(* Schneider Machine Expert - Basic project VirtualPLC_Dynamic, file version 2.6.0.0 *)
(* ProjectInformations: Name=Capstone D-03 *)
(* UserInformations: LastName=D-03, FirstName=Capstone Project *)

HARDWARE
  Cpu 0: TM221ME16R/G
  ModuleExtensionObject 0: TM3DQ8R/G
  ModuleExtensionObject 1: TM3AI8/G
  ModuleExtensionObject 2: TM3AI8/G
  EthernetConfiguration: NetworkName=M221, IpAllocationMode=FixedAddress, IpAddress=192.168.100.195, SubnetMask=255.255.255.0
  SerialLineConfiguration: Baud=Baud19200, Parity=ParityEven, DataBits=DataBits8, StopBits=StopBits1, PhysicalMedium=PhysicalMediumRs485, SlaveId=1, Addressing=SlaveAddressing
  MastTask: UsePeriodScanMode=false, PeriodScan=100
  FastTask: Period=255
  CpuBehavior: StartingMode=StartAsPreviousState, AutoSaveRamOnEeprom=true, WatchdogPeriod=250

SYMBOLS  (address, symbol, comment, settings)
  %M0       READ_GEN1
  %M1       READ_GEN2
  %M2       READ_GEN3
  %M3       READ_GEN4
  %M10      STATUS_GEN_1A_75MW
  %M11      STATUS_GEN_1B_25_MW
  %M12      STATUS_GEN_1B_75MW
  %M13      STATUS_GEN_2B_25_MW
  %M21      L101
  %M22      L201
  %M23      L303
  %M24      L304
  %M25      L305
  %M26      L401
  %M31      L301
  %M32      L302
  %M33      L402
  %M41      L403
  %M42      L404
  %M43      L405
  %M50      CONTROL_GEN1
  %M51      CONTROL_GEN2
  %M52      CONTROL_GEN3
  %M53      CONTROL_GEN4
  %M60      READ_LOAD1
  %M61      READ_LOAD2
  %M62      READ_LOAD3
  %M63      READ_LOAD4
  %M64      READ_LOAD5
  %M65      READ_LOAD6
  %M66      READ_LOAD7
  %M67      READ_LOAD8
  %M68      READ_LOAD9
  %M69      READ_LOAD10
  %M70      READ_LOAD11
  %M71      READ_LOAD12
  %MW0      SENSOR_LOAD1
  %MW1      SENSOR_LOAD2
  %MW2      SENSOR_LOAD3
  %MW3      SENSOR_LOAD4
  %MW4      SENSOR_LOAD5
  %MW5      SENSOR_LOAD6
  %MW6      SENSOR_LOAD7
  %MW7      SENSOR_LOAD8
  %MW8      SENSOR_LOAD9
  %MW9      SENSOR_LOAD10
  %MW10     SENSOR_LOAD11
  %MW11     SENSOR_LOAD12
  %MW20     JAM
  %MW21     MENIT
  %MW30     SENSOR_GEN1  "PLTA"
  %MW31     SENSOR_GEN2  "PLTS"
  %MW32     SENSOR_GEN3  "PLTGU"
  %MW33     SENSOR_GEN4  "PLTB"
  %MW54     FREQ
  %Q0.0     COIL_GEN1
  %Q0.1     COIL_GEN2
  %Q0.2     COIL_GEN3
  %Q0.3     COIL_GEN4
  %Q0.4     COIL_LOAD1
  %Q0.5     COIL_LOAD2
  %Q0.6     COIL_LOAD3
  %Q0.7     COIL_LOAD4
  %IW0.0    GEN_1_SIM  [Type=Type_0_10V, Scope=Scope_Normal, Minimum=0, Maximum=1000]
  %Q1.0     COIL_LOAD5
  %Q1.1     COIL_LOAD6
  %Q1.2     COIL_LOAD7
  %Q1.3     COIL_LOAD8
  %Q1.4     COIL_LOAD9
  %Q1.5     COIL_LOAD10
  %Q1.6     COIL_LOAD11
  %Q1.7     COIL_LOAD12

POU New POU
  (* SectionNumber=1 *)

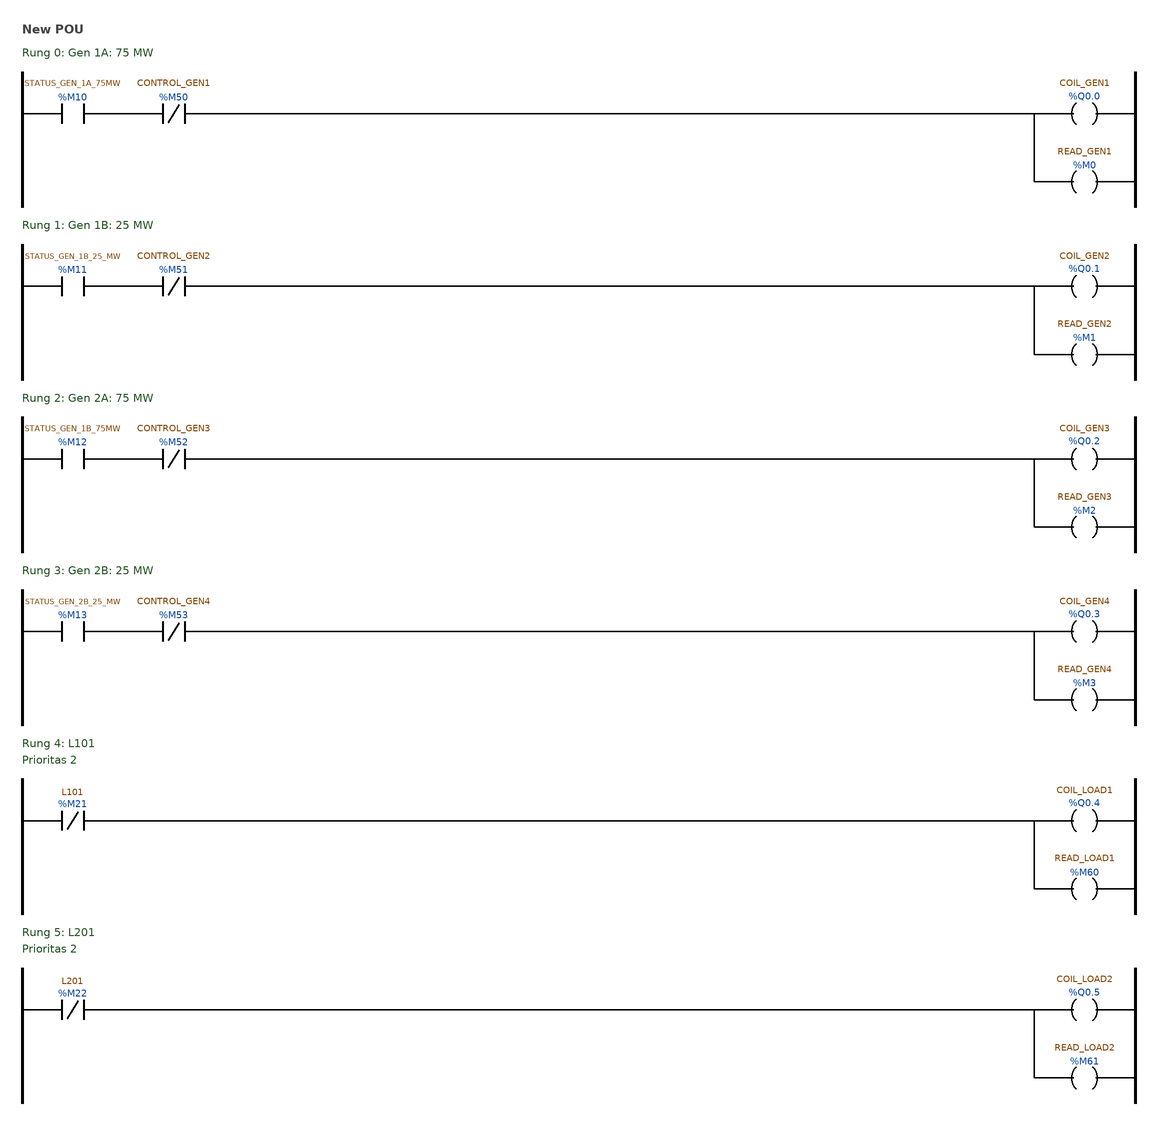

// Rung 0: Gen 1A: 75 MW
  LD %M10                 (* STATUS_GEN_1A_75MW *)
  ANDN %M50               (* CONTROL_GEN1 *)
  ST %Q0.0                (* COIL_GEN1 *)
  ST %M0                  (* READ_GEN1 *)
  // as ST:
  //   COIL_GEN1 := STATUS_GEN_1A_75MW AND NOT CONTROL_GEN1;
  //   READ_GEN1 := STATUS_GEN_1A_75MW AND NOT CONTROL_GEN1;

// Rung 1: Gen 1B: 25 MW
  LD %M11                 (* STATUS_GEN_1B_25_MW *)
  ANDN %M51               (* CONTROL_GEN2 *)
  ST %Q0.1                (* COIL_GEN2 *)
  ST %M1                  (* READ_GEN2 *)
  // as ST:
  //   COIL_GEN2 := STATUS_GEN_1B_25_MW AND NOT CONTROL_GEN2;
  //   READ_GEN2 := STATUS_GEN_1B_25_MW AND NOT CONTROL_GEN2;

// Rung 2: Gen 2A: 75 MW
  LD %M12                 (* STATUS_GEN_1B_75MW *)
  ANDN %M52               (* CONTROL_GEN3 *)
  ST %Q0.2                (* COIL_GEN3 *)
  ST %M2                  (* READ_GEN3 *)
  // as ST:
  //   COIL_GEN3 := STATUS_GEN_1B_75MW AND NOT CONTROL_GEN3;
  //   READ_GEN3 := STATUS_GEN_1B_75MW AND NOT CONTROL_GEN3;

// Rung 3: Gen 2B: 25 MW
  LD %M13                 (* STATUS_GEN_2B_25_MW *)
  ANDN %M53               (* CONTROL_GEN4 *)
  ST %Q0.3                (* COIL_GEN4 *)
  ST %M3                  (* READ_GEN4 *)
  // as ST:
  //   COIL_GEN4 := STATUS_GEN_2B_25_MW AND NOT CONTROL_GEN4;
  //   READ_GEN4 := STATUS_GEN_2B_25_MW AND NOT CONTROL_GEN4;

// Rung 4: L101
// Prioritas 2
  LDN %M21                (* L101 *)
  ST %Q0.4                (* COIL_LOAD1 *)
  ST %M60                 (* READ_LOAD1 *)
  // as ST:
  //   COIL_LOAD1 := NOT L101;
  //   READ_LOAD1 := NOT L101;

// Rung 5: L201
// Prioritas 2
  LDN %M22                (* L201 *)
  ST %Q0.5                (* COIL_LOAD2 *)
  ST %M61                 (* READ_LOAD2 *)
  // as ST:
  //   COIL_LOAD2 := NOT L201;
  //   READ_LOAD2 := NOT L201;

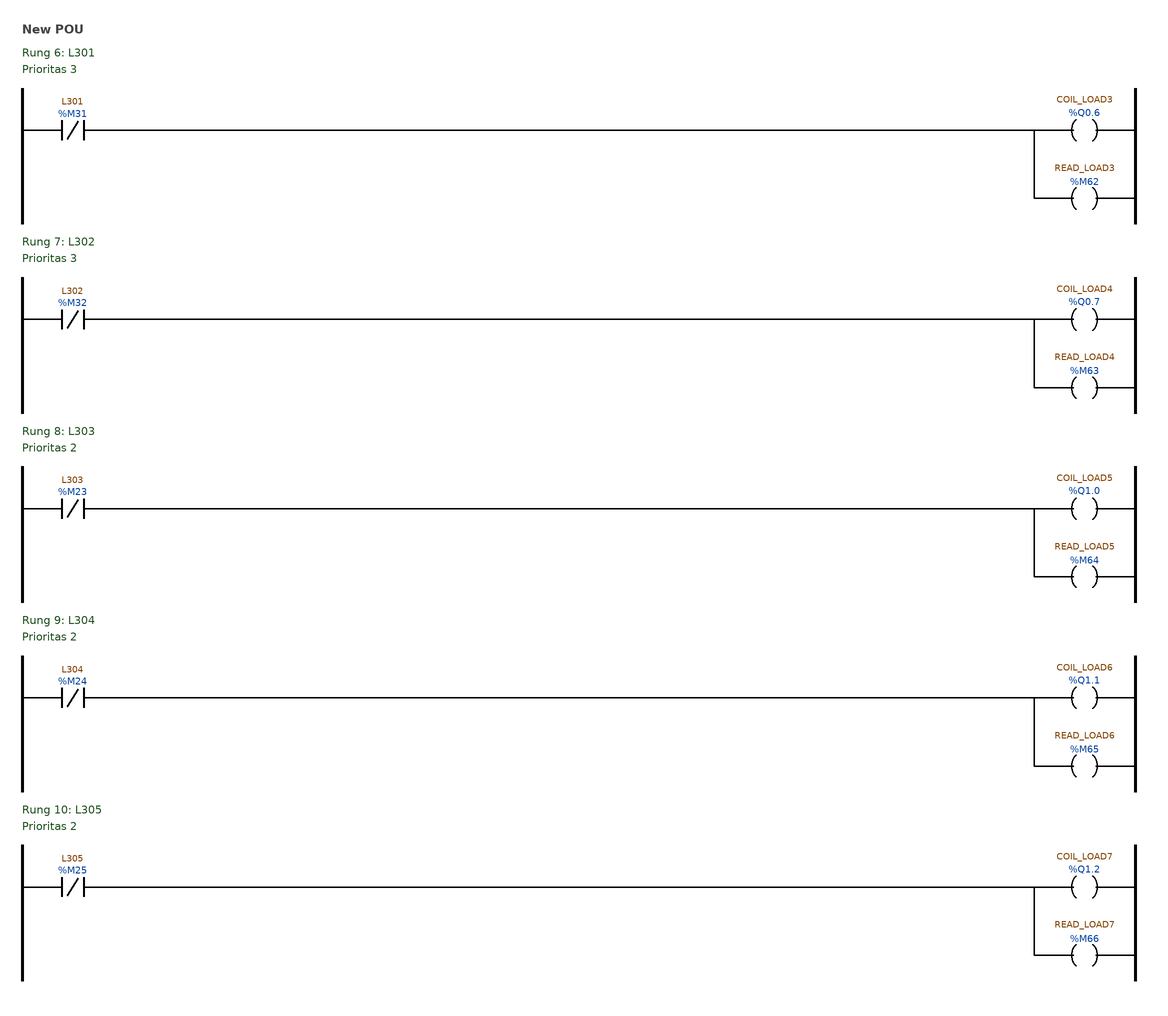

// Rung 6: L301
// Prioritas 3
  LDN %M31                (* L301 *)
  ST %Q0.6                (* COIL_LOAD3 *)
  ST %M62                 (* READ_LOAD3 *)
  // as ST:
  //   COIL_LOAD3 := NOT L301;
  //   READ_LOAD3 := NOT L301;

// Rung 7: L302
// Prioritas 3
  LDN %M32                (* L302 *)
  ST %Q0.7                (* COIL_LOAD4 *)
  ST %M63                 (* READ_LOAD4 *)
  // as ST:
  //   COIL_LOAD4 := NOT L302;
  //   READ_LOAD4 := NOT L302;

// Rung 8: L303
// Prioritas 2
  LDN %M23                (* L303 *)
  ST %Q1.0                (* COIL_LOAD5 *)
  ST %M64                 (* READ_LOAD5 *)
  // as ST:
  //   COIL_LOAD5 := NOT L303;
  //   READ_LOAD5 := NOT L303;

// Rung 9: L304
// Prioritas 2
  LDN %M24                (* L304 *)
  ST %Q1.1                (* COIL_LOAD6 *)
  ST %M65                 (* READ_LOAD6 *)
  // as ST:
  //   COIL_LOAD6 := NOT L304;
  //   READ_LOAD6 := NOT L304;

// Rung 10: L305
// Prioritas 2
  LDN %M25                (* L305 *)
  ST %Q1.2                (* COIL_LOAD7 *)
  ST %M66                 (* READ_LOAD7 *)
  // as ST:
  //   COIL_LOAD7 := NOT L305;
  //   READ_LOAD7 := NOT L305;

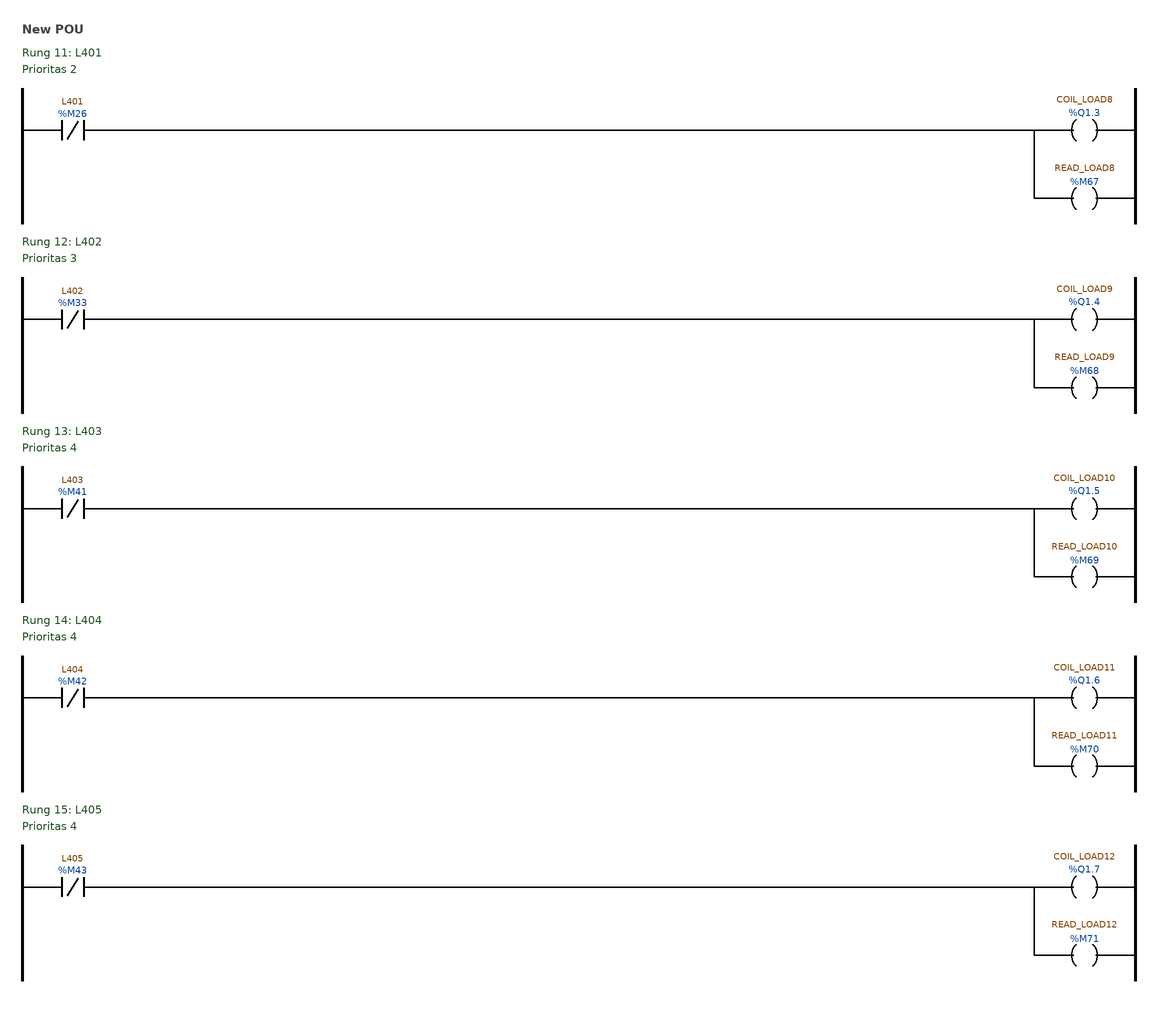

// Rung 11: L401
// Prioritas 2
  LDN %M26                (* L401 *)
  ST %Q1.3                (* COIL_LOAD8 *)
  ST %M67                 (* READ_LOAD8 *)
  // as ST:
  //   COIL_LOAD8 := NOT L401;
  //   READ_LOAD8 := NOT L401;

// Rung 12: L402
// Prioritas 3
  LDN %M33                (* L402 *)
  ST %Q1.4                (* COIL_LOAD9 *)
  ST %M68                 (* READ_LOAD9 *)
  // as ST:
  //   COIL_LOAD9 := NOT L402;
  //   READ_LOAD9 := NOT L402;

// Rung 13: L403
// Prioritas 4
  LDN %M41                (* L403 *)
  ST %Q1.5                (* COIL_LOAD10 *)
  ST %M69                 (* READ_LOAD10 *)
  // as ST:
  //   COIL_LOAD10 := NOT L403;
  //   READ_LOAD10 := NOT L403;

// Rung 14: L404
// Prioritas 4
  LDN %M42                (* L404 *)
  ST %Q1.6                (* COIL_LOAD11 *)
  ST %M70                 (* READ_LOAD11 *)
  // as ST:
  //   COIL_LOAD11 := NOT L404;
  //   READ_LOAD11 := NOT L404;

// Rung 15: L405
// Prioritas 4
  LDN %M43                (* L405 *)
  ST %Q1.7                (* COIL_LOAD12 *)
  ST %M71                 (* READ_LOAD12 *)
  // as ST:
  //   COIL_LOAD12 := NOT L405;
  //   READ_LOAD12 := NOT L405;
